// TIA Portal V20 export
TYPE "udt_BAE00TM"
   STRUCT
      PSU_Status : Bool;   // Power Supply On/Off / 电源 开/关
      Output_Drop : Bool;   // Output Drop (BDC3) / 输出 放下 (BDC3)
      Over_Temperature : Bool;   // Over Temperature (BDC2) / Over 温度 (BDC2)
      Over_Voltage : Bool;   // Over Voltage (BDC1) / Over 电压 (BDC1)
      Overload : Bool;   // Overload (BDC0) / 过载 (BDC0)
      Error_Code : Int;   // Error Code / 错误 Code
      Output_Voltage : Real;   // Output Voltage / 输出 电压
      Output_Current : Real;   // Output Current / 输出 电流
   END_STRUCT;
END_TYPE
